DATA_BLOCK "KukaRobot3_CtrlDB"
{ S7_Optimized_Access := 'FALSE' }
VERSION : 0.1
// ATTRIBUTES
// AUTO_NUMBER = False
// BLOCK_NUMBER = 2403
// END_ATTRIBUTES
"KukaRobot3_Ctrl"

BEGIN

END_DATA_BLOCK

